# EPICS autosave request: support/ip-2-10/ipApp/Db/LakeShore331.req
# FILE... LakeShore331.req
$(P)LS331:$(Q):Gain_set.VAL
$(P)LS331:$(Q):Rset_set.VAL
$(P)LS331:$(Q):Rate_set.VAL
$(P)LS331:$(Q):RampR_set.VAL
$(P)LS331:$(Q):Ramp_on.VAL
$(P)LS331:$(Q):wr_SP.VAL
$(P)LS331:$(Q):Units_sel.VAL
$(P)LS331:$(Q):Input_sel.VAL
$(P)LS331:$(Q):HeatRg.VAL
$(P)LS331:$(Q):read.SCAN
$(P)LS331:$(Q):rd_rdat_scalc.SCAN
